// TIA Portal V21 export
TYPE "ValoreAttuale"
   STRUCT
      UmCode : DInt;
      Valore : Real;
   END_STRUCT;
END_TYPE
